TYPE ST_OutputsLowLiftUnit :
(**************************************************************************************
 * 	Application		:	BoxControl Framework
 *	Revision		:	$Revision: $
 *	Revision date	:	$Date: $
 *	Last changed by	:	$Author: $
 *	URL				:	$URL: $
 *
 *	Purpose			:	Function specific outputs.
 *
 * ------------------------------------------------------------------------------------
 *	Copyright Swisslog [IP AG], Switzerland. All rights reserved.
 * 
 * ------------------------------------------------------------------------------------ 
 **************************************************************************************)	
STRUCT	
	Drive_Run_Up			: BOOL; // Drive run command lift up
	Drive_Run_Down			: BOOL; // Drive run command lift down
	Drive_Low_UpDown		: BOOL; // Drive low speed command lift
	Drive_Creep_UpDown		: BOOL; // Drive creep speed command lift	
	//Lamp_ResetLightgrid		: BOOL; // Lamp reset lightgrid	
	LowLiftEnableTransport	: BOOL; // Low lift enable transport
END_STRUCT
END_TYPE

(* stored: Version 1.1.0.1, ProductVersion 3.1.4024.4
   DUT ST_OutputsLowLiftUnit: Id {95535741-53ab-4532-b85f-cd6f6da09e68} *)
